// TIA Portal V20 export
TYPE "type_emRelations_em7"
// stored: Access Published, Namespace Unit1
   STRUCT
      "Bool" { ExternalWritable := 'False'} : Array[0..99] of Bool;
      LReal { ExternalWritable := 'False'} : Array[0..19] of LReal;
      isLinked : Bool;
      softCam : "Unit1.type_emRelations_em7_SoftCam";
      cmStatus { S7_SetPoint := 'True'} : "Unit1.type_emRelations_em7_cmStatus";
      cmConfig : Struct
         cmJRWinderAxisB : "LBC_typeAxis64PosConfiguration";
      END_STRUCT;
      sequence { S7_SetPoint := 'True'} : "Unit1.type_emRelations_em7_sequence";
   END_STRUCT;
END_TYPE
